FUNCTION_BLOCK FB_Co2FlowModelingHandler
VAR_INPUT
	valvePositionPercentage : DINT;
	pumpingPressureDelta : DINT;
	flowMeasurement : REAL;
	modelingActive : BOOL;
END_VAR
VAR_OUTPUT
	modeledOutput : LREAL;
	mF : FB_mF;
END_VAR
VAR
	u : ARRAY[1..15] OF LREAL;
	maxValveOpening : LREAL := 1.75;
	valvePosition : LREAL;
	TON_StepInterval : TON;
	firstCycle : BOOL := TRUE;
END_VAR


// Init model on first cycle
IF firstCycle THEN
	mF.setParams(
		activateObserver := TRUE);
	firstCycle := FALSE;
END_IF

// Calculate valve position
valvePosition := maxValveOpening * (TO_LREAL(valvePositionPercentage)/100);

IF modelingActive THEN
	// Fill input matrix
	u[1] := valvePosition;
	u[2] := TO_LREAL(pumpingPressureDelta);
	
	// Calculate flow every second
	TON_StepInterval(IN := TRUE, PT := T#1S);
	IF TON_StepInterval.Q THEN // AND valvePosition >= 0.25 THEN
		mF.Step(
				u := u,
				yMeas := TO_LREAL(flowMeasurement));
				
		modeledOutput := mF.y[1];
//	ELSE
//		modeledOutput := 0;
	END_IF
ELSE
	mF.Reset();
	modeledOutput := 0;
END_IF

END_FUNCTION_BLOCK

(* stored: Version 1.1.0.1, ProductVersion 3.1.4024.9
   POU FB_Co2FlowModelingHandler: Id {0c3a1a44-bbe4-40f1-bd8e-14ec8d0563a7}, SpecialFunc None *)
